// TIA Portal V20 export
TYPE "LWONIK_typePackMLStatus"
// stored: Access Published
   STRUCT
      clearing : Bool;
      stopped : Bool;
      starting : Bool;
      idle : Bool;
      suspended : Bool;
      execute : Bool;
      stopping : Bool;
      aborting : Bool;
      aborted : Bool;
      holding : Bool;
      held : Bool;
      unholding : Bool;
      suspending : Bool;
      unsuspending : Bool;
      resetting : Bool;
      completing : Bool;
      complete : Bool;
   END_STRUCT;
END_TYPE
